{attribute 'qualified_only'}
{attribute 'strict'}
{attribute 'to_string'}
TYPE E_MovementState :
(
	Idle,
	Jog,
	Halt,
	Error,
	EncHoming,
	Home
	
);
END_TYPE

(* stored: Version 1.1.0.1
   DUT E_MovementState: Id {843e2f97-5946-444b-96b3-6a820235c0ad} *)
